Staubli VAL3: CheckTraj.pgx

program CheckTraj(pointRx x_pStart (dimensions=1), pointRx x_pEnd (dimensions=1), bool& x_bTraj (dimensions=1))
  local bool l_bOk
  local joint l_jEnd
  local joint l_jStart
  local num l_nI
begin
  for l_nI=0 to 100
    pTraj.trsf=interpolateL(x_pStart.trsf,x_pEnd.trsf,l_nI/100)
    if l_nI==0
      l_jStart=herej()
    else
      l_jStart=l_jEnd
    endIf
    l_bOk=pointToJoint(tTool,l_jStart,pTraj,l_jEnd)

    if l_bOk==false
      x_bTraj=false
      call ListPop("CantMove")
      return
    endIf
  endFor
  x_bTraj=true
end
